Fanuc KAREL source: kt00749.KL

-- PROVISIONAL review KL for V770-1; original PC SHA256 ffdb1bae37030792426dc9a207e2cab6e7a087bdda87709e6cb6c767e3663c75
-- Incomplete behavior may be omitted. Consult companion uncertainty JSON. Do not deploy.
PROGRAM KT00749
%NOLOCKGROUP
VAR
  I1 : INTEGER
  I2 : INTEGER
  OUT : REAL
BEGIN
  -- UNRESOLVED_PC offsets 5-16; opcodes 2E,23
  -- UNRESOLVED_PC offsets 21-32; opcodes 2E,23
  -- UNRESOLVED_PC offsets 37-48; opcodes 2E,23
  -- UNRESOLVED_PC offsets 53-64; opcodes 2E,23
  -- UNRESOLVED_PC offsets 69-83; opcodes 21,50,64,23
  -- UNRESOLVED_PC offsets 88-92; opcodes 7F
END KT00749
